// TIA Portal V20 export
// export: Created 2025-12-01T14:56:09.5415812Z, ExportSetting None, DisplayName Totally Integrated Automation Portal, DisplayVersion V20 Update 3, DisplayName TIA Portal Openness, DisplayVersion V20 Update 3, DisplayName TIA Portal Version Control Interface, DisplayVersion V20 Update 3, DisplayName STEP 7 Professional, DisplayVersion V20 Update 3, DisplayName STEP 7 Safety, DisplayVersion V20 Update 2, DisplayName WinCC Basic/Comfort/Advanced, DisplayVersion V20 Update 3, DisplayName WinCC Professional, DisplayVersion V20 Update 3, DisplayName WinCC Unified, DisplayVersion V20 Update 3
TYPE "FUDT_Marcas_ciclo_seguridad"
// stored: IsFailsafeCompliant true
   STRUCT
      "0_1_seg" { ExternalAccessible := 'False'; ExternalVisible := 'False'; ExternalWritable := 'False'} : Bool;
      "0_2_seg" : Bool;
      "0_4_seg" : Bool;
      "0_5_seg" : Bool;
      "0_8_seg" : Bool;
      "1_seg" : Bool;
      "1_6_seg" : Bool;
      "2_seg" : Bool;
   END_STRUCT;
END_TYPE
